Fanuc KAREL source: IO0195.KL

-- PROVISIONAL review KL for V940-1; original PC SHA256 461f186fc26cfec4827c166ee1f44e194eae12e18ed16b18e83fb14bfa5345fd
-- Incomplete behavior may be omitted. Consult companion uncertainty JSON. Do not deploy.
PROGRAM IO0195
%NOLOCKGROUP
-- UNRESOLVED_LOCAL_POOL 5 cells at code offset 13; source declarations unknown
-- DIRECT_LOCAL_WORD_ACCESS alone does not prove INTEGER, REAL, or BOOLEAN
BEGIN
  -- V9_ZERO_TABLE_METADATA_HINT layout=0002_ascii; no indexed target words; source/name/runtime held
  -- UNRESOLVED_PC offsets 0-18; opcodes 2B,2C,7B
  -- UNRESOLVED_PC offsets 23-30; opcodes 9D,23
  -- UNRESOLVED_PC offsets 35-49; opcodes 2E,22,9D,33,35
  -- UNRESOLVED_PC offsets 54-61; opcodes 9D,23
  -- UNRESOLVED_PC offsets 66-77; opcodes 2E,23
  -- UNRESOLVED_PC offsets 82-108; opcodes 27,27,9D,22,27,9D,31,7E,4A
  -- UNRESOLVED_PC offsets 113-129; opcodes 22,32,34,23
  -- UNRESOLVED_PC offsets 134-138; opcodes 7F
  -- UNRESOLVED_PC offsets 143-147; opcodes 27,AA
  -- UNRESOLVED_PC offsets 152-156; opcodes 7F
END IO0195
